FUNCTION_BLOCK Empty EXTENDS CraneMovement
VAR_INPUT
END_VAR
VAR_OUTPUT
END_VAR
VAR
END_VAR

SUPER^(
	iPalletsInRack:=iPalletsInRack,
	aSlots:=aSlots,
	fioOutputs:=fioOutputs,
	sCurrentOperation:=sCurrentOperation);
	
IF bStart 
	AND iStep = 0
	AND iPalletsInRack > 0
	THEN
	iStep := 10;
	bBusy := TRUE;
ELSIF NOT bStart
	THEN
	bDone := FALSE;
	bBusy := FALSE;
	iStep := 0;
END_IF


CASE iStep OF
	

	10: // Go to required position
	
		sCurrentOperation := Concat('Going to slot position ', INT_TO_STRING(iSlotPosition));
		fioOutputs.iSCPosition := iSlotPosition;
		motionTimer.IN := TRUE;
		
		IF NOT fioInputs.bSCMovingX
			 AND NOT fioInputs.bSCMovingZ
			 AND motionTimer.Q
			 THEN
			 
			 motionTimer.IN := FALSE;
			 iStep := 20; 
		END_IF
		
	20: // load the pallet on the stacker crane
		sCurrentOperation := 'Loading';
		fioOutputs.bSCLeft := TRUE;
		IF fioInputs.bSCLeftLimit
			THEN
			istep := 30;
		END_IF
		
	30: // Lift 
	
		fioOutputs.bSCLift := TRUE;
		liftTimer.IN := TRUE;
		
		IF liftTimer.Q
			THEN
			liftTimer.IN := FALSE;
			iStep := 40;
		END_IF
		
	40: // Stacker crane in middle position
	
		fioOutputs.bSCLeft := FALSE;
		IF fioInputs.bSCMiddlLimit
			THEN
			istep := 50;
		END_IF	
		
	50: // Lower the crane
	
		fioOutputs.bSCLift := FALSE;
		liftTimer.IN := TRUE;
		
		IF liftTimer.Q
			THEN
			aSlots[iSlotPosition] := FALSE;
			iPalletsInRack:=iPalletsInRack-1;
			liftTimer.IN := FALSE;
			iStep := 60;
		END_IF
	
		
	60: // Return to the load position
		sCurrentOperation := 'Return to initial position';

		fioOutputs.iSCPosition := 55;
		motionTimer.IN := TRUE;
		
		IF NOT fioInputs.bSCMovingX
			 AND NOT fioInputs.bSCMovingZ
			 AND motionTimer.Q
			 THEN
			 motionTimer.IN := FALSE;
			
			 iStep := 70; 
		END_IF
		
	70: // Lift the stacker crane
	
		fioOutputs.bSCLift := TRUE;
		liftTimer.IN := TRUE;
		
		IF liftTimer.Q
			THEN
			liftTimer.IN := FALSE;
			iStep := 80;
		END_IF
		
	80: // Start loading pallet on the stacker crane 
	
		fioOutputs.bSCLeft := TRUE;
		IF fioInputs.bSCLeftLimit 
			THEN
			iStep := 90;
		END_IF	
		
	90: // Lower stacker crane
		
		fioOutputs.bSCLift := FALSE;
		liftTimer.IN := TRUE;
		
		IF liftTimer.Q
			THEN
			liftTimer.IN := FALSE;
			iStep := 100;
		END_IF	
		
	100: // Return to the middle position
		fioOutputs.bSCLeft := FALSE;
		IF fioInputs.bSCMiddlLimit
			THEN
			bDone := TRUE;
			bBusy := FALSE;
			istep := 110;
		END_IF		

END_CASE

END_FUNCTION_BLOCK

(* stored: Version 1.1.0.1, ProductVersion 3.1.4024.10
   POU Empty: Id {24fefab1-b201-4437-8aaf-9aa4a1c43b4a}, SpecialFunc None *)
